{attribute 'qualified_only'}
VAR_GLOBAL
	MasterUid				: ULINT := 999999999;
	VisualisationReady		: BOOL;
	VisualisationHeartbeatCounter	: ULINT;
	DeviceCount				: UINT;
	SnapshotUpdateCounter	: ULINT;
	SnapshotTimestamp		: ULINT;
	Devices					: ARRAY [0..63] OF EspDeviceSnapshot;
END_VAR

(* stored: Version 1.1.0.1
   GVL GVL_EspVisualisation: Id {7d60281c-c9c9-4dcb-a516-a8835df66c66} *)
